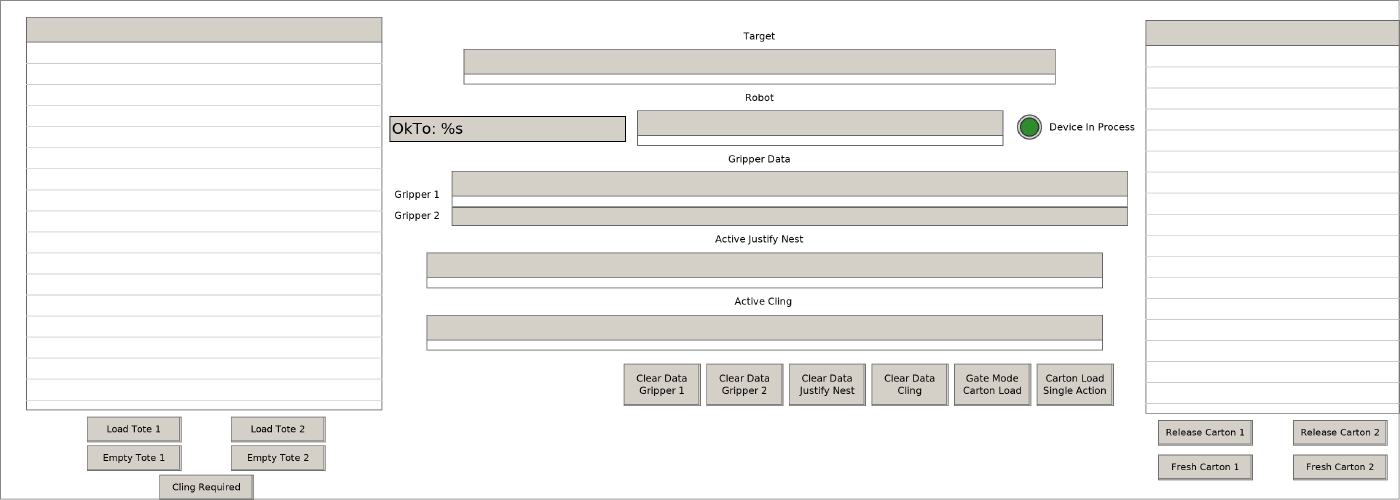
VISUALIZATION PartTracking  // 1661x594
    Table (31,20 422x467), data array: Stn100_06_CartonLoadMain.fbCartonLoadMain.pToteSpur[Stn100_06_CartonLoadMain.fbCartonLoadMain.Act.Target.Tote]^.SpurTote.Slots_RS
        p3854506369: Stn100_06_CartonLoadMain.fbCartonLoadMain.pToteSpur[Stn100_06_CartonLoadMain.fbCartonLoadMain.Act.Target.Tote]^.SpurTote.Slots_RS[INDEX].Row
        p1892666644: Stn100_06_CartonLoadMain.fbCartonLoadMain.pToteSpur[Stn100_06_CartonLoadMain.fbCartonLoadMain.Act.Target.Tote]^.SpurTote.Slots_RS[INDEX].Column
        p338671338: Stn100_06_CartonLoadMain.fbCartonLoadMain.pToteSpur[Stn100_06_CartonLoadMain.fbCartonLoadMain.Act.Target.Tote]^.SpurTote.Slots_RS[INDEX].DeviceSN
        p2170511999: Stn100_06_CartonLoadMain.fbCartonLoadMain.pToteSpur[Stn100_06_CartonLoadMain.fbCartonLoadMain.Act.Target.Tote]^.SpurTote.Slots_RS[INDEX].Length
        p3723444502: Stn100_06_CartonLoadMain.fbCartonLoadMain.pToteSpur[Stn100_06_CartonLoadMain.fbCartonLoadMain.Act.Target.Tote]^.SpurTote.Slots_RS[INDEX].Width
        p1218418051: Stn100_06_CartonLoadMain.fbCartonLoadMain.pToteSpur[Stn100_06_CartonLoadMain.fbCartonLoadMain.Act.Target.Tote]^.SpurTote.Slots_RS[INDEX].Height
        p746581629: Stn100_06_CartonLoadMain.fbCartonLoadMain.pToteSpur[Stn100_06_CartonLoadMain.fbCartonLoadMain.Act.Target.Tote]^.SpurTote.Slots_RS[INDEX].WMOrderID
        p3104783080: Stn100_06_CartonLoadMain.fbCartonLoadMain.pToteSpur[Stn100_06_CartonLoadMain.fbCartonLoadMain.Act.Target.Tote]^.SpurTote.Slots_RS[INDEX].CartonNum
    Rectangle (789,101 224x30), "Robot"
    Table (506,300 802x42), data array: Stn100_06_CartonLoadMain.fbCartonLoadMain.pJustifyNest[Stn100_06_CartonLoadMain.fbCartonLoadMain.Act.Target.JustifyNest]^.Device
        p3854506369: Stn100_06_CartonLoadMain.fbCartonLoadMain.pJustifyNest[Stn100_06_CartonLoadMain.fbCartonLoadMain.Act.Target.JustifyNest]^.Device.Justified
        p1892666644: Stn100_06_CartonLoadMain.fbCartonLoadMain.pJustifyNest[Stn100_06_CartonLoadMain.fbCartonLoadMain.Act.Target.JustifyNest]^.Device.ClingRequired
        p338671338: Stn100_06_CartonLoadMain.fbCartonLoadMain.pJustifyNest[Stn100_06_CartonLoadMain.fbCartonLoadMain.Act.Target.JustifyNest]^.Device.ClingSize
        p2170511999: Stn100_06_CartonLoadMain.fbCartonLoadMain.pJustifyNest[Stn100_06_CartonLoadMain.fbCartonLoadMain.Act.Target.JustifyNest]^.Device.CartonNum
        p3723444502: Stn100_06_CartonLoadMain.fbCartonLoadMain.pJustifyNest[Stn100_06_CartonLoadMain.fbCartonLoadMain.Act.Target.JustifyNest]^.Device.ToteRFID
        p1218418051: Stn100_06_CartonLoadMain.fbCartonLoadMain.pJustifyNest[Stn100_06_CartonLoadMain.fbCartonLoadMain.Act.Target.JustifyNest]^.Device.ToteSide
        p746581629: Stn100_06_CartonLoadMain.fbCartonLoadMain.pJustifyNest[Stn100_06_CartonLoadMain.fbCartonLoadMain.Act.Target.JustifyNest]^.Device.JustifyNest
        p3104783080: Stn100_06_CartonLoadMain.fbCartonLoadMain.pJustifyNest[Stn100_06_CartonLoadMain.fbCartonLoadMain.Act.Target.JustifyNest]^.Device.Heading
        p2501879983: Stn100_06_CartonLoadMain.fbCartonLoadMain.pJustifyNest[Stn100_06_CartonLoadMain.fbCartonLoadMain.Act.Target.JustifyNest]^.Device.SN
        p7306298: Stn100_06_CartonLoadMain.fbCartonLoadMain.pJustifyNest[Stn100_06_CartonLoadMain.fbCartonLoadMain.Act.Target.JustifyNest]^.Device.Status
        p1933151965: Stn100_06_CartonLoadMain.fbCartonLoadMain.pJustifyNest[Stn100_06_CartonLoadMain.fbCartonLoadMain.Act.Target.JustifyNest]^.Device.XPOStatus
        p3863566920: Stn100_06_CartonLoadMain.fbCartonLoadMain.pJustifyNest[Stn100_06_CartonLoadMain.fbCartonLoadMain.Act.Target.JustifyNest]^.Device.Route
        p2192122294: Stn100_06_CartonLoadMain.fbCartonLoadMain.pJustifyNest[Stn100_06_CartonLoadMain.fbCartonLoadMain.Act.Target.JustifyNest]^.Device.RMRoute
        p400160035: Stn100_06_CartonLoadMain.fbCartonLoadMain.pJustifyNest[Stn100_06_CartonLoadMain.fbCartonLoadMain.Act.Target.JustifyNest]^.Device.SKU
        p1265227338: Stn100_06_CartonLoadMain.fbCartonLoadMain.pJustifyNest[Stn100_06_CartonLoadMain.fbCartonLoadMain.Act.Target.JustifyNest]^.Device.PuckSide
        p3726181087: Stn100_06_CartonLoadMain.fbCartonLoadMain.pJustifyNest[Stn100_06_CartonLoadMain.fbCartonLoadMain.Act.Target.JustifyNest]^.Device.Length
        p3136911649: Stn100_06_CartonLoadMain.fbCartonLoadMain.pJustifyNest[Stn100_06_CartonLoadMain.fbCartonLoadMain.Act.Target.JustifyNest]^.Device.Width
        p797552052: Stn100_06_CartonLoadMain.fbCartonLoadMain.pJustifyNest[Stn100_06_CartonLoadMain.fbCartonLoadMain.Act.Target.JustifyNest]^.Device.Height
        p60375027: Stn100_06_CartonLoadMain.fbCartonLoadMain.pJustifyNest[Stn100_06_CartonLoadMain.fbCartonLoadMain.Act.Target.JustifyNest]^.Device.Size
        p2531912550: Stn100_06_CartonLoadMain.fbCartonLoadMain.pJustifyNest[Stn100_06_CartonLoadMain.fbCartonLoadMain.Act.Target.JustifyNest]^.Device.IsHighPriority
        p693678525: Stn100_06_CartonLoadMain.fbCartonLoadMain.pJustifyNest[Stn100_06_CartonLoadMain.fbCartonLoadMain.Act.Target.JustifyNest]^.Device.RowaTrayType
        p3156763944: Stn100_06_CartonLoadMain.fbCartonLoadMain.pJustifyNest[Stn100_06_CartonLoadMain.fbCartonLoadMain.Act.Target.JustifyNest]^.Device.EvalData
        p511219082: Cling Req
        p1755163831: Cling Size
    Rectangle (789,269 224x30), "Active Justify Nest"
    Table (506,374 802x42), data array: Stn100_06_CartonLoadMain.fbCartonLoadMain.ClingDevice[Stn100_06_CartonLoadMain.fbCartonLoadMain.Act.Target.Cling]
        p3854506369: Stn100_06_CartonLoadMain.fbCartonLoadMain.ClingDevice[Stn100_06_CartonLoadMain.fbCartonLoadMain.Act.Target.Cling].Justified
        p1892666644: Stn100_06_CartonLoadMain.fbCartonLoadMain.ClingDevice[Stn100_06_CartonLoadMain.fbCartonLoadMain.Act.Target.Cling].ClingRequired
        p338671338: Stn100_06_CartonLoadMain.fbCartonLoadMain.ClingDevice[Stn100_06_CartonLoadMain.fbCartonLoadMain.Act.Target.Cling].ClingSize
        p2170511999: Stn100_06_CartonLoadMain.fbCartonLoadMain.ClingDevice[Stn100_06_CartonLoadMain.fbCartonLoadMain.Act.Target.Cling].CartonNum
        p3723444502: Stn100_06_CartonLoadMain.fbCartonLoadMain.ClingDevice[Stn100_06_CartonLoadMain.fbCartonLoadMain.Act.Target.Cling].ToteRFID
        p1218418051: Stn100_06_CartonLoadMain.fbCartonLoadMain.ClingDevice[Stn100_06_CartonLoadMain.fbCartonLoadMain.Act.Target.Cling].ToteSide
        p746581629: Stn100_06_CartonLoadMain.fbCartonLoadMain.ClingDevice[Stn100_06_CartonLoadMain.fbCartonLoadMain.Act.Target.Cling].JustifyNest
        p3104783080: Stn100_06_CartonLoadMain.fbCartonLoadMain.ClingDevice[Stn100_06_CartonLoadMain.fbCartonLoadMain.Act.Target.Cling].Heading
        p2501879983: Stn100_06_CartonLoadMain.fbCartonLoadMain.ClingDevice[Stn100_06_CartonLoadMain.fbCartonLoadMain.Act.Target.Cling].SN
        p7306298: Stn100_06_CartonLoadMain.fbCartonLoadMain.ClingDevice[Stn100_06_CartonLoadMain.fbCartonLoadMain.Act.Target.Cling].Status
        p1933151965: Stn100_06_CartonLoadMain.fbCartonLoadMain.ClingDevice[Stn100_06_CartonLoadMain.fbCartonLoadMain.Act.Target.Cling].XPOStatus
        p3863566920: Stn100_06_CartonLoadMain.fbCartonLoadMain.ClingDevice[Stn100_06_CartonLoadMain.fbCartonLoadMain.Act.Target.Cling].Route
        p2192122294: Stn100_06_CartonLoadMain.fbCartonLoadMain.ClingDevice[Stn100_06_CartonLoadMain.fbCartonLoadMain.Act.Target.Cling].RMRoute
        p400160035: Stn100_06_CartonLoadMain.fbCartonLoadMain.ClingDevice[Stn100_06_CartonLoadMain.fbCartonLoadMain.Act.Target.Cling].SKU
        p1265227338: Stn100_06_CartonLoadMain.fbCartonLoadMain.ClingDevice[Stn100_06_CartonLoadMain.fbCartonLoadMain.Act.Target.Cling].PuckSide
        p3726181087: Stn100_06_CartonLoadMain.fbCartonLoadMain.ClingDevice[Stn100_06_CartonLoadMain.fbCartonLoadMain.Act.Target.Cling].Length
        p3136911649: Stn100_06_CartonLoadMain.fbCartonLoadMain.ClingDevice[Stn100_06_CartonLoadMain.fbCartonLoadMain.Act.Target.Cling].Width
        p797552052: Stn100_06_CartonLoadMain.fbCartonLoadMain.ClingDevice[Stn100_06_CartonLoadMain.fbCartonLoadMain.Act.Target.Cling].Height
        p60375027: Stn100_06_CartonLoadMain.fbCartonLoadMain.ClingDevice[Stn100_06_CartonLoadMain.fbCartonLoadMain.Act.Target.Cling].Size
        p2531912550: Stn100_06_CartonLoadMain.fbCartonLoadMain.ClingDevice[Stn100_06_CartonLoadMain.fbCartonLoadMain.Act.Target.Cling].IsHighPriority
        p693678525: Stn100_06_CartonLoadMain.fbCartonLoadMain.ClingDevice[Stn100_06_CartonLoadMain.fbCartonLoadMain.Act.Target.Cling].RowaTrayType
        p3156763944: Stn100_06_CartonLoadMain.fbCartonLoadMain.ClingDevice[Stn100_06_CartonLoadMain.fbCartonLoadMain.Act.Target.Cling].EvalData
        p511219082: Cling Req
        p1755163831: Cling Size
    Rectangle (794,343 224x30), "Active Cling"
    Table (1359,24 302x467), data array: Stn100_06_CartonLoadMain.fbCartonLoadMain.pCartonNest[Stn100_06_CartonLoadMain.fbCartonLoadMain.Act.Target.Carton]^.Carton.RecordSet
        p3104783080: Stn100_06_CartonLoadMain.fbCartonLoadMain.CartonDevice[].RecordSet
        p2501879983: Stn100_06_CartonLoadMain.fbCartonLoadMain.CartonDevice[].RecordSetSize
        p3854506369: Stn100_06_CartonLoadMain.fbCartonLoadMain.pCartonNest[Stn100_06_CartonLoadMain.fbCartonLoadMain.Act.Target.Carton]^.Carton.RecordSet[INDEX].Row
        p1892666644: Stn100_06_CartonLoadMain.fbCartonLoadMain.pCartonNest[Stn100_06_CartonLoadMain.fbCartonLoadMain.Act.Target.Carton]^.Carton.RecordSet[INDEX].Column
        p338671338: Stn100_06_CartonLoadMain.fbCartonLoadMain.pCartonNest[Stn100_06_CartonLoadMain.fbCartonLoadMain.Act.Target.Carton]^.Carton.RecordSet[INDEX].DeviceSN
        p1755163831: Serial Number
    Table (550,58 702x42), data array: Stn100_06_CartonLoadMain.fbCartonLoadMain.Act.Target
        p3854506369: Stn100_06_CartonLoadMain.fbCartonLoadMain.Act.Target.RobotCmd
        p1892666644: Stn100_06_CartonLoadMain.fbCartonLoadMain.Act.Target.RobotGripper
        p338671338: Stn100_06_CartonLoadMain.fbCartonLoadMain.Act.Target.Tote
        p2170511999: Stn100_06_CartonLoadMain.fbCartonLoadMain.Act.Target.ToteSlot
        p3723444502: Stn100_06_CartonLoadMain.fbCartonLoadMain.Act.Target.ToteRow
        p1218418051: Stn100_06_CartonLoadMain.fbCartonLoadMain.Act.Target.ToteColumn
        p746581629: Stn100_06_CartonLoadMain.fbCartonLoadMain.Act.Target.Carton
        p3104783080: Stn100_06_CartonLoadMain.fbCartonLoadMain.Act.Target.CartonSlot
        p2501879983: Stn100_06_CartonLoadMain.fbCartonLoadMain.Act.Target.CartonRow
        p7306298: Stn100_06_CartonLoadMain.fbCartonLoadMain.Act.Target.CartonColumn
        p1933151965: Stn100_06_CartonLoadMain.fbCartonLoadMain.Act.Target.JustifyNest
        p3863566920: Stn100_06_CartonLoadMain.fbCartonLoadMain.Act.Target.Cling
        p2192122294: Stn100_06_CartonLoadMain.fbCartonLoadMain.ClingDevice[Stn100_06_CartonLoadMain.fbCartonLoadMain.Act.Target.Cling].RMRoute
        p400160035: Stn100_06_CartonLoadMain.fbCartonLoadMain.ClingDevice[Stn100_06_CartonLoadMain.fbCartonLoadMain.Act.Target.Cling].SKU
        p1265227338: Stn100_06_CartonLoadMain.fbCartonLoadMain.ClingDevice[Stn100_06_CartonLoadMain.fbCartonLoadMain.Act.Target.Cling].PuckSide
        p3726181087: Stn100_06_CartonLoadMain.fbCartonLoadMain.ClingDevice[Stn100_06_CartonLoadMain.fbCartonLoadMain.Act.Target.Cling].Length
        p3136911649: Stn100_06_CartonLoadMain.fbCartonLoadMain.ClingDevice[Stn100_06_CartonLoadMain.fbCartonLoadMain.Act.Target.Cling].Width
        p797552052: Stn100_06_CartonLoadMain.fbCartonLoadMain.ClingDevice[Stn100_06_CartonLoadMain.fbCartonLoadMain.Act.Target.Cling].Height
        p60375027: Stn100_06_CartonLoadMain.fbCartonLoadMain.ClingDevice[Stn100_06_CartonLoadMain.fbCartonLoadMain.Act.Target.Cling].Size
        p2531912550: Stn100_06_CartonLoadMain.fbCartonLoadMain.ClingDevice[Stn100_06_CartonLoadMain.fbCartonLoadMain.Act.Target.Cling].IsHighPriority
        p693678525: Stn100_06_CartonLoadMain.fbCartonLoadMain.ClingDevice[Stn100_06_CartonLoadMain.fbCartonLoadMain.Act.Target.Cling].RowaTrayType
        p3156763944: Stn100_06_CartonLoadMain.fbCartonLoadMain.ClingDevice[Stn100_06_CartonLoadMain.fbCartonLoadMain.Act.Target.Cling].EvalData
    Table (756,131 434x42), data array: Stn100_06_CartonLoadMain.fbCartonLoadMain.pRobot^
        p3854506369: Stn100_06_CartonLoadMain.fbCartonLoadMain.pRobot^.Framework
        p1892666644: Stn100_06_CartonLoadMain.fbCartonLoadMain.pRobot^.Cmd
        p338671338: Stn100_06_CartonLoadMain.fbCartonLoadMain.pRobot^.Rsp
        p2170511999: Stn100_06_CartonLoadMain.fbCartonLoadMain.pRobot^.Index
        p3723444502: Stn100_06_CartonLoadMain.fbCartonLoadMain.pRobot^.AuxIndex
        p1218418051: Stn100_06_CartonLoadMain.fbCartonLoadMain.pRobot^.Angle
        p746581629: Stn100_06_CartonLoadMain.fbCartonLoadMain.pRobot^.XOffset
        p3104783080: Stn100_06_CartonLoadMain.fbCartonLoadMain.pRobot^.YOffset
        p2501879983: Stn100_06_CartonLoadMain.fbCartonLoadMain.pRobot^.ZOffset
        p7306298: Stn100_06_CartonLoadMain.fbCartonLoadMain.pRobot^.ApproachOnly
        p1933151965: Stn100_06_CartonLoadMain.fbCartonLoadMain.pRobot^.GeneralOutput
        p3863566920: Stn100_06_CartonLoadMain.fbCartonLoadMain.pRobot^.GeneralInput
        p2192122294: Stn100_06_CartonLoadMain.fbCartonLoadMain.pRobot^.GripperInputStatus
        p400160035: Stn100_06_CartonLoadMain.fbCartonLoadMain.pRobot^.InZone
        p1265227338: Stn100_06_CartonLoadMain.fbCartonLoadMain.pRobot^.ZoneAccessGranted
        p3726181087: Stn100_06_CartonLoadMain.fbCartonLoadMain.pRobot^.ZoneAccessReq
        p3136911649: Stn100_06_CartonLoadMain.fbCartonLoadMain.pRobot^.OtherDeviceInZone
        p797552052: Stn100_06_CartonLoadMain.fbCartonLoadMain.pRobot^.OtherDeviceHeartbeat
        p60375027: Stn100_06_CartonLoadMain.fbCartonLoadMain.pRobot^.AccessReqFromOtherDevice
        p2531912550: Stn100_06_CartonLoadMain.fbCartonLoadMain.pRobot^.AccessGrantedFromOtherDevice
    Button (1374,499 112x30), "Release Carton 1"
        tap Stn100_06_CartonLoadMain.fbCartonLoadMain.ReleaseCarton[1]
    Button (1534,499 112x30), "Release Carton 2"
        tap Stn100_06_CartonLoadMain.fbCartonLoadMain.ReleaseCarton[2]
    Lamp1 (1203,134 37x34), variable: Stn100_06_CartonLoadMain.fbTC.fbTC01.DevicesInProcess, style: Lamp-Lamp1-Green
    Rectangle (1242,136 110x30), "Device In Process"
    Button (103,495 112x30), "Load Tote 1"
        tap Stn100_21_ToteSpur1.fbToteSpur.Debug_LoadData
    Button (274,495 112x30), "Load Tote 2"
        tap Stn100_22_ToteSpur2.fbToteSpur.Debug_LoadData
    Button (740,432 91x50), "Clear Data Gripper 1"
        toggle Stn100_06_CartonLoadMain.fbCartonLoadMain.Debug_ClearRobotGrip1Data
    Button (936,432 91x50), "Clear Data Justify Nest"
        toggle Stn100_06_CartonLoadMain.fbCartonLoadMain.Debug_ClearJustifyNestData
    Button (1034,432 91x50), "Clear Data Cling"
        toggle Stn100_06_CartonLoadMain.fbCartonLoadMain.Debug_ClearClingData
    Button (1132,432 91x50), "Gate Mode Carton Load", colour toggle: Stn100_06_CartonLoadMain.fbCartonLoadMain.Debug_GateActionMode
        p573394764: Green
        toggle Stn100_06_CartonLoadMain.fbCartonLoadMain.Debug_GateActionMode
    Button (838,432 91x50), "Clear Data Gripper 2"
        toggle Stn100_06_CartonLoadMain.fbCartonLoadMain.Debug_ClearRobotGrip2Data
    Table (536,203 802x42), data array: Stn100_06_CartonLoadMain.fbCartonLoadMain.RobotDevice[1]
        p3854506369: Stn100_06_CartonLoadMain.fbCartonLoadMain.RobotDevice[1].Justified
        p1892666644: Stn100_06_CartonLoadMain.fbCartonLoadMain.RobotDevice[1].ClingRequired
        p338671338: Stn100_06_CartonLoadMain.fbCartonLoadMain.RobotDevice[1].ClingSize
        p2170511999: Stn100_06_CartonLoadMain.fbCartonLoadMain.RobotDevice[1].CartonNum
        p3723444502: Stn100_06_CartonLoadMain.fbCartonLoadMain.RobotDevice[1].ToteRFID
        p1218418051: Stn100_06_CartonLoadMain.fbCartonLoadMain.RobotDevice[1].ToteSide
        p746581629: Stn100_06_CartonLoadMain.fbCartonLoadMain.RobotDevice[1].JustifyNest
        p3104783080: Stn100_06_CartonLoadMain.fbCartonLoadMain.RobotDevice[1].Heading
        p2501879983: Stn100_06_CartonLoadMain.fbCartonLoadMain.RobotDevice[1].SN
        p7306298: Stn100_06_CartonLoadMain.fbCartonLoadMain.RobotDevice[1].Status
        p1933151965: Stn100_06_CartonLoadMain.fbCartonLoadMain.RobotDevice[1].XPOStatus
        p3863566920: Stn100_06_CartonLoadMain.fbCartonLoadMain.RobotDevice[1].Route
        p2192122294: Stn100_06_CartonLoadMain.fbCartonLoadMain.RobotDevice[1].RMRoute
        p400160035: Stn100_06_CartonLoadMain.fbCartonLoadMain.RobotDevice[1].SKU
        p1265227338: Stn100_06_CartonLoadMain.fbCartonLoadMain.RobotDevice[1].PuckSide
        p3726181087: Stn100_06_CartonLoadMain.fbCartonLoadMain.RobotDevice[1].Length
        p3136911649: Stn100_06_CartonLoadMain.fbCartonLoadMain.RobotDevice[1].Width
        p797552052: Stn100_06_CartonLoadMain.fbCartonLoadMain.RobotDevice[1].Height
        p60375027: Stn100_06_CartonLoadMain.fbCartonLoadMain.RobotDevice[1].Size
        p2531912550: Stn100_06_CartonLoadMain.fbCartonLoadMain.RobotDevice[1].IsHighPriority
        p693678525: Stn100_06_CartonLoadMain.fbCartonLoadMain.RobotDevice[1].RowaTrayType
        p3156763944: Stn100_06_CartonLoadMain.fbCartonLoadMain.RobotDevice[1].EvalData
        p511219082: Cling Req
    Rectangle (789,174 224x30), "Gripper Data"
    Rectangle (455,216 80x30), "Gripper 1"
    Rectangle (455,241 80x30), "Gripper 2"
    Table (536,246 802x22), data array: Stn100_06_CartonLoadMain.fbCartonLoadMain.RobotDevice[2]
        p3854506369: Stn100_06_CartonLoadMain.fbCartonLoadMain.RobotDevice[2].Justified
        p1892666644: Stn100_06_CartonLoadMain.fbCartonLoadMain.RobotDevice[2].ClingRequired
        p338671338: Stn100_06_CartonLoadMain.fbCartonLoadMain.RobotDevice[2].ClingSize
        p2170511999: Stn100_06_CartonLoadMain.fbCartonLoadMain.RobotDevice[2].CartonNum
        p3723444502: Stn100_06_CartonLoadMain.fbCartonLoadMain.RobotDevice[2].ToteRFID
        p1218418051: Stn100_06_CartonLoadMain.fbCartonLoadMain.RobotDevice[2].ToteSide
        p746581629: Stn100_06_CartonLoadMain.fbCartonLoadMain.RobotDevice[2].JustifyNest
        p3104783080: Stn100_06_CartonLoadMain.fbCartonLoadMain.RobotDevice[2].Heading
        p2501879983: Stn100_06_CartonLoadMain.fbCartonLoadMain.RobotDevice[2].SN
        p7306298: Stn100_06_CartonLoadMain.fbCartonLoadMain.RobotDevice[2].Status
        p1933151965: Stn100_06_CartonLoadMain.fbCartonLoadMain.RobotDevice[2].XPOStatus
        p3863566920: Stn100_06_CartonLoadMain.fbCartonLoadMain.RobotDevice[2].Route
        p2192122294: Stn100_06_CartonLoadMain.fbCartonLoadMain.RobotDevice[2].RMRoute
        p400160035: Stn100_06_CartonLoadMain.fbCartonLoadMain.RobotDevice[2].SKU
        p1265227338: Stn100_06_CartonLoadMain.fbCartonLoadMain.RobotDevice[2].PuckSide
        p3726181087: Stn100_06_CartonLoadMain.fbCartonLoadMain.RobotDevice[2].Length
        p3136911649: Stn100_06_CartonLoadMain.fbCartonLoadMain.RobotDevice[2].Width
        p797552052: Stn100_06_CartonLoadMain.fbCartonLoadMain.RobotDevice[2].Height
        p60375027: Stn100_06_CartonLoadMain.fbCartonLoadMain.RobotDevice[2].Size
        p2531912550: Stn100_06_CartonLoadMain.fbCartonLoadMain.RobotDevice[2].IsHighPriority
        p693678525: Stn100_06_CartonLoadMain.fbCartonLoadMain.RobotDevice[2].RowaTrayType
        p3156763944: Stn100_06_CartonLoadMain.fbCartonLoadMain.RobotDevice[2].EvalData
        p511219082: Cling Req
        p1755163831: Cling Size
    Button (1230,432 91x50), "Carton Load Single Action", colour toggle: Stn100_06_CartonLoadMain.fbCartonLoadMain.Debug_SingleGateAction
        p573394764: Green
        toggle Stn100_06_CartonLoadMain.fbCartonLoadMain.Debug_SingleGateAction
    Rectangle (462,138 280x30), "OkTo: %s", text variable: Stn100_06_CartonLoadMain.fbTC.Act.OkTo, colour toggle: Stn100_06_CartonLoadMain.fbTC.Act.OkTo > 0, text index: cCartonLoadMainOkTo
    Button (1374,540 112x30), "Fresh Carton 1"
        tap Stn100_35_CartonNest1.fbCartonNest.Debug_FreshCarton
    Button (1534,540 112x30), "Fresh Carton 2"
        tap Stn100_36_CartonNest2.fbCartonNest.Debug_FreshCarton
    Button (189,564 112x30), "Cling Required", colour toggle: Stn100_06_CartonLoadMain.fbCartonLoadMain.Debug_ClingRequired
        p2175578022: White
        toggle Stn100_06_CartonLoadMain.fbCartonLoadMain.Debug_ClingRequired
    Button (103,529 112x30), "Empty Tote 1"
        tap Stn100_21_ToteSpur1.fbToteSpur.Debug_EmptyTote
    Button (274,529 112x30), "Empty Tote 2"
        tap Stn100_22_ToteSpur2.fbToteSpur.Debug_EmptyTote
    Rectangle (789,28 224x30), "Target"
END_VISUALIZATION

(* stored: Version 1.1.0.1, ProductVersion 3.1.4024.6
   Visu PartTracking: Id {4d92c097-37dc-41e7-85bb-b24c769a7bf1} *)
